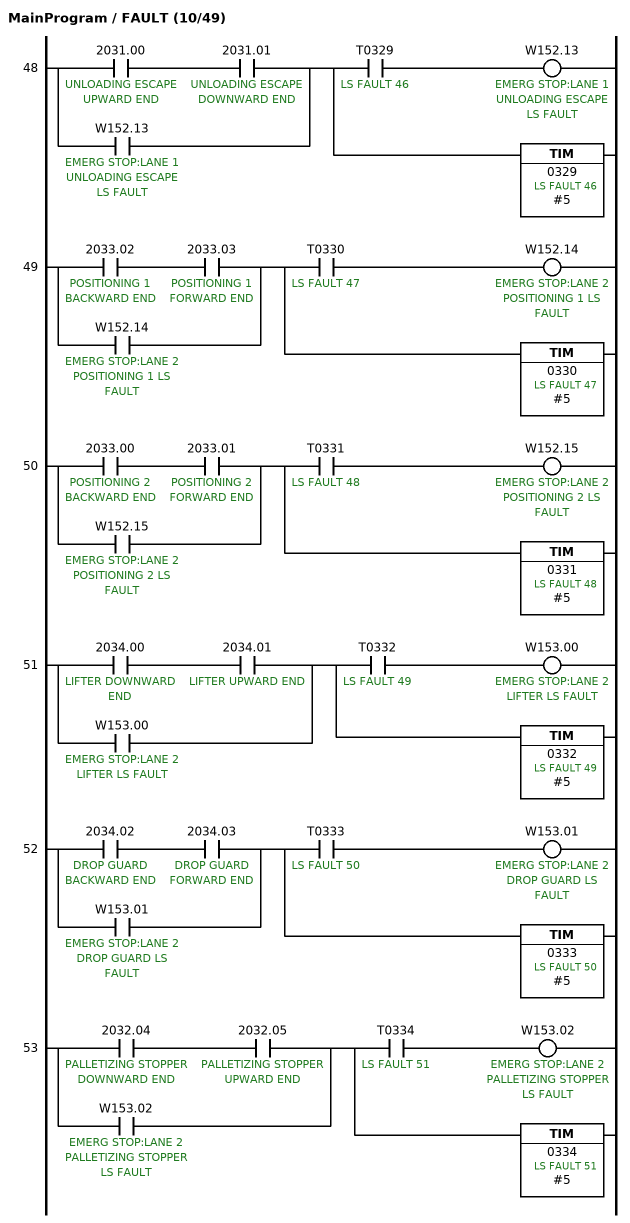
; [picture p72: MainProgram / FAULT, rungs 48-53]
; rung 48
LD 2031.00  ; UNLOADING ESCAPE UPWARD END
AND 2031.01  ; UNLOADING ESCAPE DOWNWARD END
OR W152.13  ; EMERG STOP:LANE 1 UNLOADING ESCAPE LS FAULT
OUT TR0
AND T0329  ; LS FAULT 46
OUT W152.13  ; EMERG STOP:LANE 1 UNLOADING ESCAPE LS FAULT
LD TR0
TIM 0329 #5  ; LS FAULT 46
; rung 49
LD 2033.02  ; POSITIONING 1 BACKWARD END
AND 2033.03  ; POSITIONING 1 FORWARD END
OR W152.14  ; EMERG STOP:LANE 2 POSITIONING 1 LS FAULT
OUT TR0
AND T0330  ; LS FAULT 47
OUT W152.14  ; EMERG STOP:LANE 2 POSITIONING 1 LS FAULT
LD TR0
TIM 0330 #5  ; LS FAULT 47
; rung 50
LD 2033.00  ; POSITIONING 2 BACKWARD END
AND 2033.01  ; POSITIONING 2 FORWARD END
OR W152.15  ; EMERG STOP:LANE 2 POSITIONING 2 LS FAULT
OUT TR0
AND T0331  ; LS FAULT 48
OUT W152.15  ; EMERG STOP:LANE 2 POSITIONING 2 LS FAULT
LD TR0
TIM 0331 #5  ; LS FAULT 48
; rung 51
LD 2034.00  ; LIFTER DOWNWARD END
AND 2034.01  ; LIFTER UPWARD END
OR W153.00  ; EMERG STOP:LANE 2 LIFTER LS FAULT
OUT TR0
AND T0332  ; LS FAULT 49
OUT W153.00  ; EMERG STOP:LANE 2 LIFTER LS FAULT
LD TR0
TIM 0332 #5  ; LS FAULT 49
; rung 52
LD 2034.02  ; DROP GUARD BACKWARD END
AND 2034.03  ; DROP GUARD FORWARD END
OR W153.01  ; EMERG STOP:LANE 2 DROP GUARD LS FAULT
OUT TR0
AND T0333  ; LS FAULT 50
OUT W153.01  ; EMERG STOP:LANE 2 DROP GUARD LS FAULT
LD TR0
TIM 0333 #5  ; LS FAULT 50
; rung 53
LD 2032.04  ; PALLETIZING STOPPER DOWNWARD END
AND 2032.05  ; PALLETIZING STOPPER UPWARD END
OR W153.02  ; EMERG STOP:LANE 2 PALLETIZING STOPPER LS FAULT
OUT TR0
AND T0334  ; LS FAULT 51
OUT W153.02  ; EMERG STOP:LANE 2 PALLETIZING STOPPER LS FAULT
LD TR0
TIM 0334 #5  ; LS FAULT 51

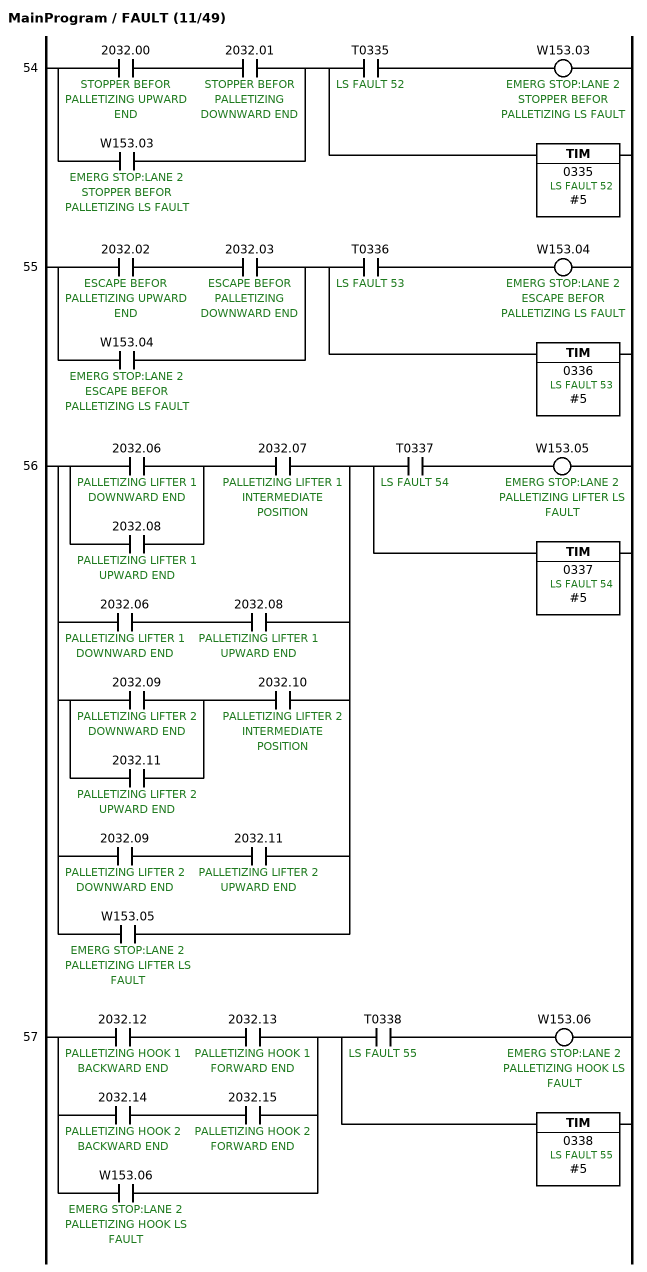
; rung 54
LD 2032.00  ; STOPPER BEFOR PALLETIZING UPWARD END
AND 2032.01  ; STOPPER BEFOR PALLETIZING DOWNWARD END
OR W153.03  ; EMERG STOP:LANE 2 STOPPER BEFOR PALLETIZING LS FAULT
OUT TR0
AND T0335  ; LS FAULT 52
OUT W153.03  ; EMERG STOP:LANE 2 STOPPER BEFOR PALLETIZING LS FAULT
LD TR0
TIM 0335 #5  ; LS FAULT 52
; rung 55
LD 2032.02  ; ESCAPE BEFOR PALLETIZING UPWARD END
AND 2032.03  ; ESCAPE BEFOR PALLETIZING DOWNWARD END
OR W153.04  ; EMERG STOP:LANE 2 ESCAPE BEFOR PALLETIZING LS FAULT
OUT TR0
AND T0336  ; LS FAULT 53
OUT W153.04  ; EMERG STOP:LANE 2 ESCAPE BEFOR PALLETIZING LS FAULT
LD TR0
TIM 0336 #5  ; LS FAULT 53
; rung 56
LD 2032.06  ; PALLETIZING LIFTER 1 DOWNWARD END
OR 2032.08  ; PALLETIZING LIFTER 1 UPWARD END
AND 2032.07  ; PALLETIZING LIFTER 1 INTERMEDIATE POSITION
LD 2032.06  ; PALLETIZING LIFTER 1 DOWNWARD END
AND 2032.08  ; PALLETIZING LIFTER 1 UPWARD END
ORLD
LD 2032.09  ; PALLETIZING LIFTER 2 DOWNWARD END
OR 2032.11  ; PALLETIZING LIFTER 2 UPWARD END
AND 2032.10  ; PALLETIZING LIFTER 2 INTERMEDIATE POSITION
ORLD
LD 2032.09  ; PALLETIZING LIFTER 2 DOWNWARD END
AND 2032.11  ; PALLETIZING LIFTER 2 UPWARD END
ORLD
OR W153.05  ; EMERG STOP:LANE 2 PALLETIZING LIFTER LS FAULT
OUT TR0
AND T0337  ; LS FAULT 54
OUT W153.05  ; EMERG STOP:LANE 2 PALLETIZING LIFTER LS FAULT
LD TR0
TIM 0337 #5  ; LS FAULT 54
; rung 57
LD 2032.12  ; PALLETIZING HOOK 1 BACKWARD END
AND 2032.13  ; PALLETIZING HOOK 1 FORWARD END
LD 2032.14  ; PALLETIZING HOOK 2 BACKWARD END
AND 2032.15  ; PALLETIZING HOOK 2 FORWARD END
ORLD
OR W153.06  ; EMERG STOP:LANE 2 PALLETIZING HOOK LS FAULT
OUT TR0
AND T0338  ; LS FAULT 55
OUT W153.06  ; EMERG STOP:LANE 2 PALLETIZING HOOK LS FAULT
LD TR0
TIM 0338 #5  ; LS FAULT 55

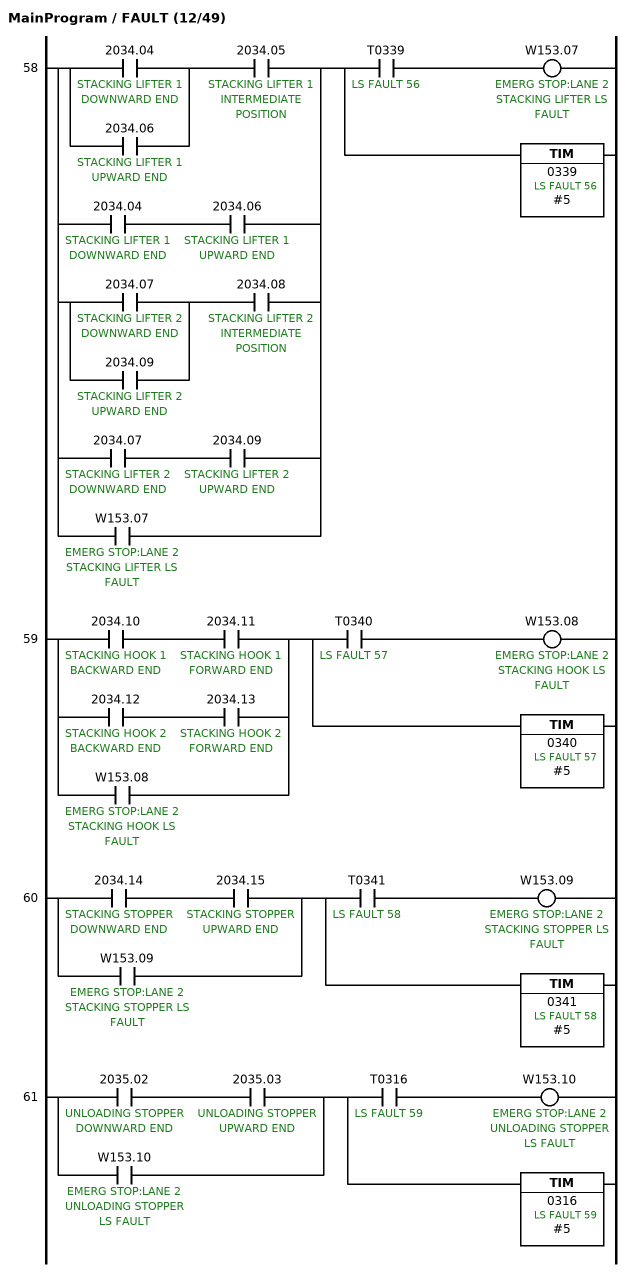
; rung 58
LD 2034.04  ; STACKING LIFTER 1 DOWNWARD END
OR 2034.06  ; STACKING LIFTER 1 UPWARD END
AND 2034.05  ; STACKING LIFTER 1 INTERMEDIATE POSITION
LD 2034.04  ; STACKING LIFTER 1 DOWNWARD END
AND 2034.06  ; STACKING LIFTER 1 UPWARD END
ORLD
LD 2034.07  ; STACKING LIFTER 2 DOWNWARD END
OR 2034.09  ; STACKING LIFTER 2 UPWARD END
AND 2034.08  ; STACKING LIFTER 2 INTERMEDIATE POSITION
ORLD
LD 2034.07  ; STACKING LIFTER 2 DOWNWARD END
AND 2034.09  ; STACKING LIFTER 2 UPWARD END
ORLD
OR W153.07  ; EMERG STOP:LANE 2 STACKING LIFTER LS FAULT
OUT TR0
AND T0339  ; LS FAULT 56
OUT W153.07  ; EMERG STOP:LANE 2 STACKING LIFTER LS FAULT
LD TR0
TIM 0339 #5  ; LS FAULT 56
; rung 59
LD 2034.10  ; STACKING HOOK 1 BACKWARD END
AND 2034.11  ; STACKING HOOK 1 FORWARD END
LD 2034.12  ; STACKING HOOK 2 BACKWARD END
AND 2034.13  ; STACKING HOOK 2 FORWARD END
ORLD
OR W153.08  ; EMERG STOP:LANE 2 STACKING HOOK LS FAULT
OUT TR0
AND T0340  ; LS FAULT 57
OUT W153.08  ; EMERG STOP:LANE 2 STACKING HOOK LS FAULT
LD TR0
TIM 0340 #5  ; LS FAULT 57
; rung 60
LD 2034.14  ; STACKING STOPPER DOWNWARD END
AND 2034.15  ; STACKING STOPPER UPWARD END
OR W153.09  ; EMERG STOP:LANE 2 STACKING STOPPER LS FAULT
OUT TR0
AND T0341  ; LS FAULT 58
OUT W153.09  ; EMERG STOP:LANE 2 STACKING STOPPER LS FAULT
LD TR0
TIM 0341 #5  ; LS FAULT 58
; rung 61
LD 2035.02  ; UNLOADING STOPPER DOWNWARD END
AND 2035.03  ; UNLOADING STOPPER UPWARD END
OR W153.10  ; EMERG STOP:LANE 2 UNLOADING STOPPER LS FAULT
OUT TR0
AND T0316  ; LS FAULT 59
OUT W153.10  ; EMERG STOP:LANE 2 UNLOADING STOPPER LS FAULT
LD TR0
TIM 0316 #5  ; LS FAULT 59

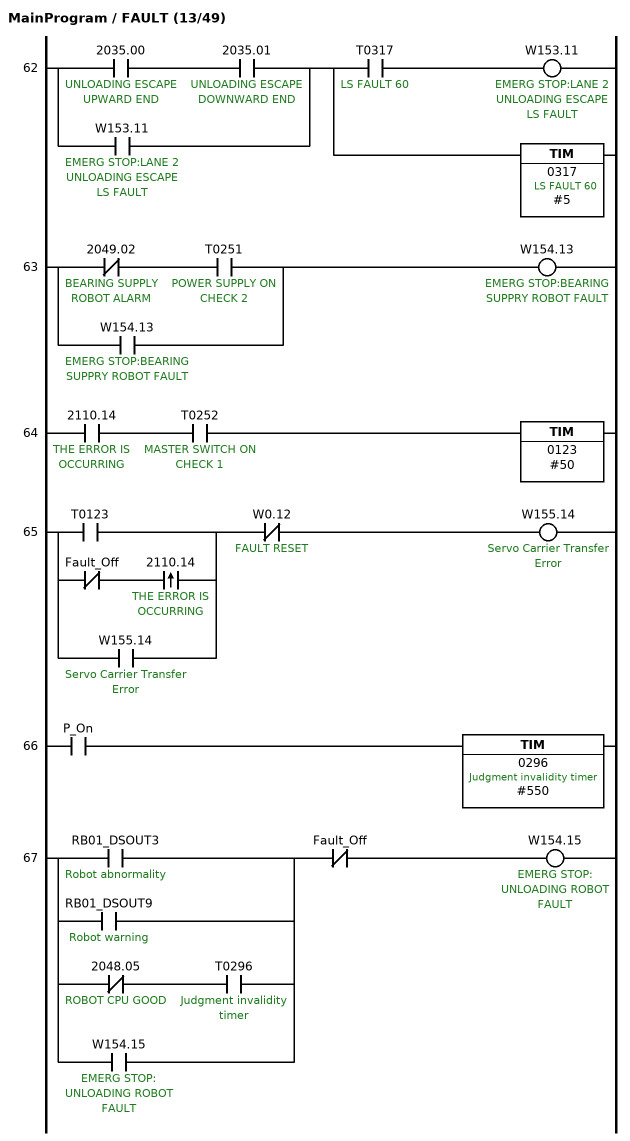
; rung 62
LD 2035.00  ; UNLOADING ESCAPE UPWARD END
AND 2035.01  ; UNLOADING ESCAPE DOWNWARD END
OR W153.11  ; EMERG STOP:LANE 2 UNLOADING ESCAPE LS FAULT
OUT TR0
AND T0317  ; LS FAULT 60
OUT W153.11  ; EMERG STOP:LANE 2 UNLOADING ESCAPE LS FAULT
LD TR0
TIM 0317 #5  ; LS FAULT 60
; rung 63
LDNOT 2049.02  ; BEARING SUPPLY ROBOT ALARM
AND T0251  ; POWER SUPPLY ON CHECK 2
OR W154.13  ; EMERG STOP:BEARING SUPPRY ROBOT FAULT
OUT W154.13  ; EMERG STOP:BEARING SUPPRY ROBOT FAULT
; rung 64
LD 2110.14  ; THE ERROR IS OCCURRING
AND T0252  ; MASTER SWITCH ON CHECK 1
TIM 0123 #50
; rung 65
LD T0123
LDNOT Fault_Off
@AND 2110.14  ; THE ERROR IS OCCURRING
ORLD
OR W155.14  ; Servo Carrier Transfer Error
ANDNOT W0.12  ; FAULT RESET
OUT W155.14  ; Servo Carrier Transfer Error
; rung 66
LD P_On
TIM 0296 #550  ; Judgment invalidity timer
; rung 67
LD RB01_DSOUT3  ; Robot abnormality
OR RB01_DSOUT9  ; Robot warning
LDNOT 2048.05  ; ROBOT CPU GOOD
AND T0296  ; Judgment invalidity timer
ORLD
OR W154.15  ; EMERG STOP:UNLOADING ROBOT FAULT
ANDNOT Fault_Off
OUT W154.15  ; EMERG STOP:UNLOADING ROBOT FAULT

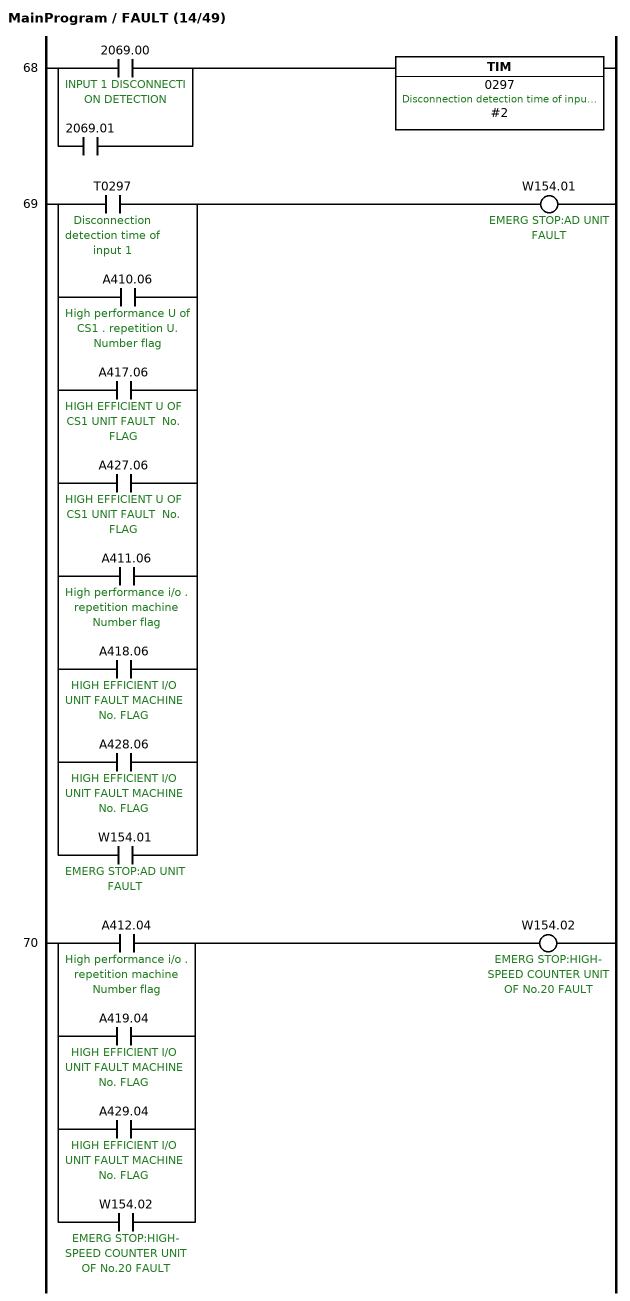
; rung 68
LD 2069.00  ; INPUT 1 DISCONNECTION DETECTION
OR 2069.01
TIM 0297 #2  ; Disconnection detection time of input 1
; rung 69
LD T0297  ; Disconnection detection time of input 1
OR A410.06  ; High performance U of CS1 . repetition U. Number flag
OR A417.06  ; HIGH EFFICIENT U OF CS1 UNIT FAULT  No. FLAG
OR A427.06  ; HIGH EFFICIENT U OF CS1 UNIT FAULT  No. FLAG
OR A411.06  ; High performance i/o . repetition machine Number flag
OR A418.06  ; HIGH EFFICIENT I/O UNIT FAULT MACHINE No. FLAG
OR A428.06  ; HIGH EFFICIENT I/O UNIT FAULT MACHINE No. FLAG
OR W154.01  ; EMERG STOP:AD UNIT FAULT
OUT W154.01  ; EMERG STOP:AD UNIT FAULT
; rung 70
LD A412.04  ; High performance i/o . repetition machine Number flag
OR A419.04  ; HIGH EFFICIENT I/O UNIT FAULT MACHINE No. FLAG
OR A429.04  ; HIGH EFFICIENT I/O UNIT FAULT MACHINE No. FLAG
OR W154.02  ; EMERG STOP:HIGH-SPEED COUNTER UNIT OF No.20 FAULT
OUT W154.02  ; EMERG STOP:HIGH-SPEED COUNTER UNIT OF No.20 FAULT

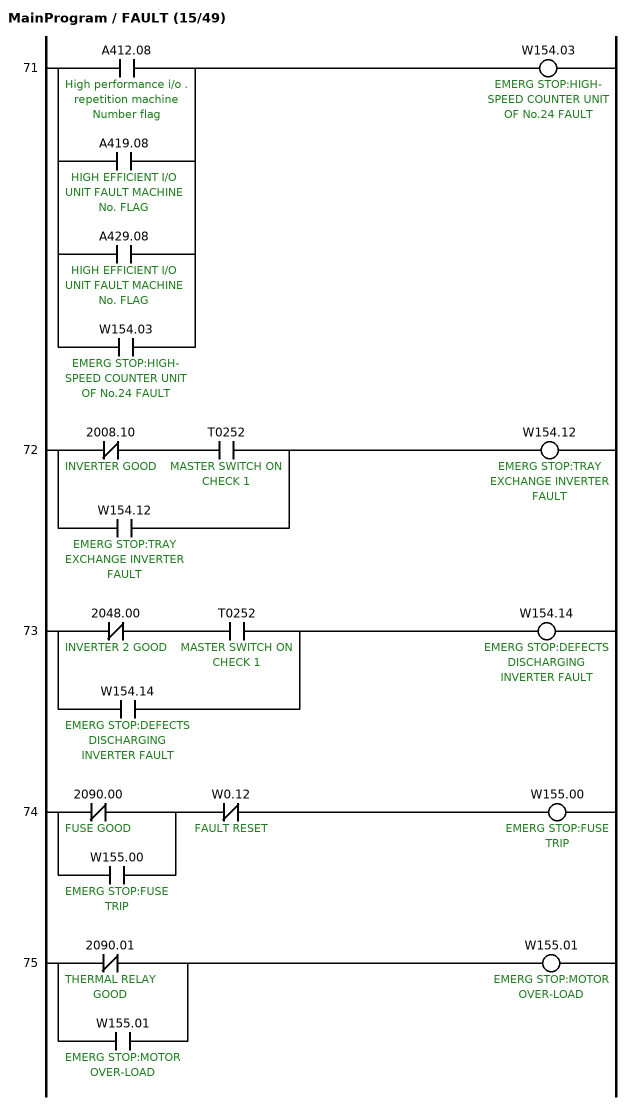
; rung 71
LD A412.08  ; High performance i/o . repetition machine Number flag
OR A419.08  ; HIGH EFFICIENT I/O UNIT FAULT MACHINE No. FLAG
OR A429.08  ; HIGH EFFICIENT I/O UNIT FAULT MACHINE No. FLAG
OR W154.03  ; EMERG STOP:HIGH-SPEED COUNTER UNIT OF No.24 FAULT
OUT W154.03  ; EMERG STOP:HIGH-SPEED COUNTER UNIT OF No.24 FAULT
; rung 72
LDNOT 2008.10  ; INVERTER GOOD
AND T0252  ; MASTER SWITCH ON CHECK 1
OR W154.12  ; EMERG STOP:TRAY EXCHANGE INVERTER FAULT
OUT W154.12  ; EMERG STOP:TRAY EXCHANGE INVERTER FAULT
; rung 73
LDNOT 2048.00  ; INVERTER 2 GOOD
AND T0252  ; MASTER SWITCH ON CHECK 1
OR W154.14  ; EMERG STOP:DEFECTS DISCHARGING INVERTER FAULT
OUT W154.14  ; EMERG STOP:DEFECTS DISCHARGING INVERTER FAULT
; rung 74
LDNOT 2090.00  ; FUSE GOOD
OR W155.00  ; EMERG STOP:FUSE TRIP
ANDNOT W0.12  ; FAULT RESET
OUT W155.00  ; EMERG STOP:FUSE TRIP
; rung 75
LDNOT 2090.01  ; THERMAL RELAY GOOD
OR W155.01  ; EMERG STOP:MOTOR OVER-LOAD
OUT W155.01  ; EMERG STOP:MOTOR OVER-LOAD

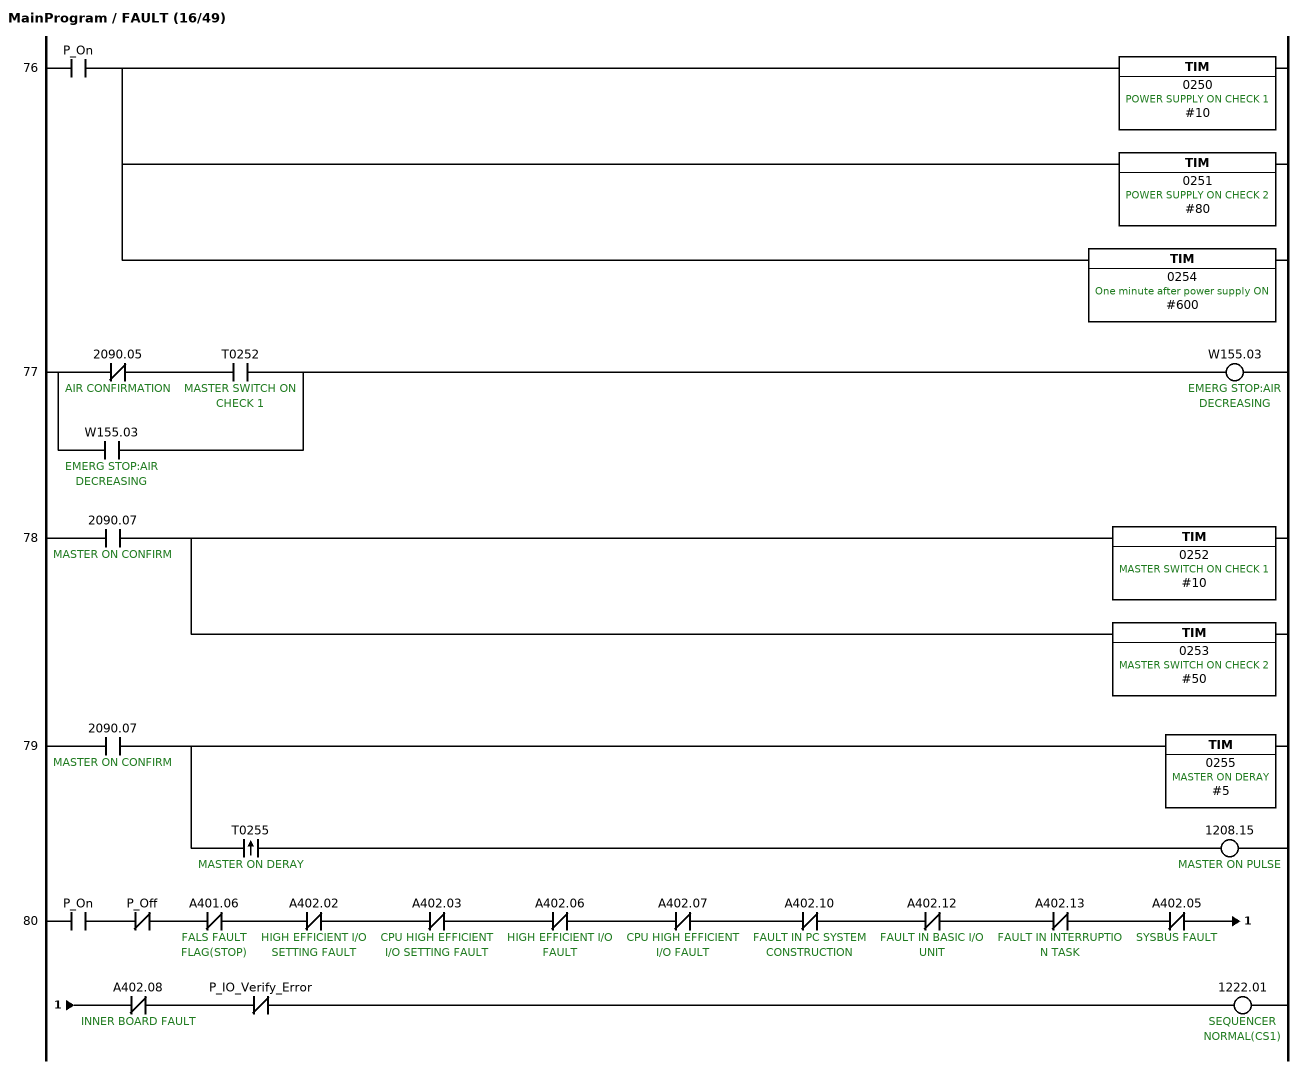
; rung 76
LD P_On
TIM 0250 #10  ; POWER SUPPLY ON CHECK 1
TIM 0251 #80  ; POWER SUPPLY ON CHECK 2
TIM 0254 #600  ; One minute after power supply ON
; rung 77
LDNOT 2090.05  ; AIR CONFIRMATION
AND T0252  ; MASTER SWITCH ON CHECK 1
OR W155.03  ; EMERG STOP:AIR DECREASING
OUT W155.03  ; EMERG STOP:AIR DECREASING
; rung 78
LD 2090.07  ; MASTER ON CONFIRM
TIM 0252 #10  ; MASTER SWITCH ON CHECK 1
TIM 0253 #50  ; MASTER SWITCH ON CHECK 2
; rung 79
LD 2090.07  ; MASTER ON CONFIRM
TIM 0255 #5  ; MASTER ON DERAY
@AND T0255  ; MASTER ON DERAY
OUT 1208.15  ; MASTER ON PULSE
; rung 80
LD P_On
ANDNOT P_Off
ANDNOT A401.06  ; FALS FAULT FLAG(STOP)
ANDNOT A402.02  ; HIGH EFFICIENT I/O SETTING FAULT
ANDNOT A402.03  ; CPU HIGH EFFICIENT I/O SETTING FAULT
ANDNOT A402.06  ; HIGH EFFICIENT I/O FAULT
ANDNOT A402.07  ; CPU HIGH EFFICIENT I/O FAULT
ANDNOT A402.10  ; FAULT IN PC SYSTEM CONSTRUCTION
ANDNOT A402.12  ; FAULT IN BASIC I/O UNIT
ANDNOT A402.13  ; FAULT IN INTERRUPTION TASK
ANDNOT A402.05  ; SYSBUS FAULT
ANDNOT A402.08  ; INNER BOARD FAULT
ANDNOT P_IO_Verify_Error
OUT 1222.01  ; SEQUENCER NORMAL(CS1)

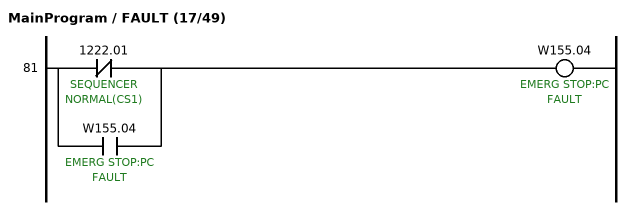
; rung 81
LDNOT 1222.01  ; SEQUENCER NORMAL(CS1)
OR W155.04  ; EMERG STOP:PC FAULT
OUT W155.04  ; EMERG STOP:PC FAULT

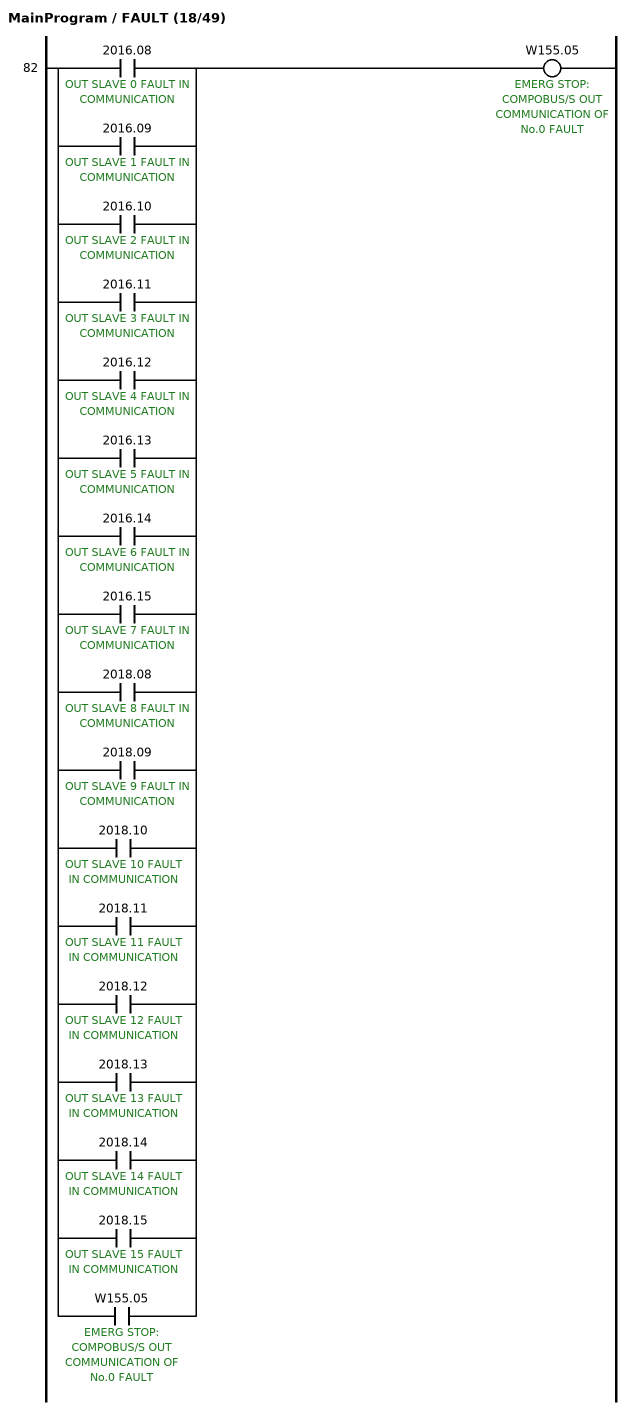
; rung 82
LD 2016.08  ; OUT SLAVE 0 FAULT IN COMMUNICATION
OR 2016.09  ; OUT SLAVE 1 FAULT IN COMMUNICATION
OR 2016.10  ; OUT SLAVE 2 FAULT IN COMMUNICATION
OR 2016.11  ; OUT SLAVE 3 FAULT IN COMMUNICATION
OR 2016.12  ; OUT SLAVE 4 FAULT IN COMMUNICATION
OR 2016.13  ; OUT SLAVE 5 FAULT IN COMMUNICATION
OR 2016.14  ; OUT SLAVE 6 FAULT IN COMMUNICATION
OR 2016.15  ; OUT SLAVE 7 FAULT IN COMMUNICATION
OR 2018.08  ; OUT SLAVE 8 FAULT IN COMMUNICATION
OR 2018.09  ; OUT SLAVE 9 FAULT IN COMMUNICATION
OR 2018.10  ; OUT SLAVE 10 FAULT IN COMMUNICATION
OR 2018.11  ; OUT SLAVE 11 FAULT IN COMMUNICATION
OR 2018.12  ; OUT SLAVE 12 FAULT IN COMMUNICATION
OR 2018.13  ; OUT SLAVE 13 FAULT IN COMMUNICATION
OR 2018.14  ; OUT SLAVE 14 FAULT IN COMMUNICATION
OR 2018.15  ; OUT SLAVE 15 FAULT IN COMMUNICATION
OR W155.05  ; EMERG STOP:COMPOBUS/S OUT COMMUNICATION OF No.0 FAULT
OUT W155.05  ; EMERG STOP:COMPOBUS/S OUT COMMUNICATION OF No.0 FAULT

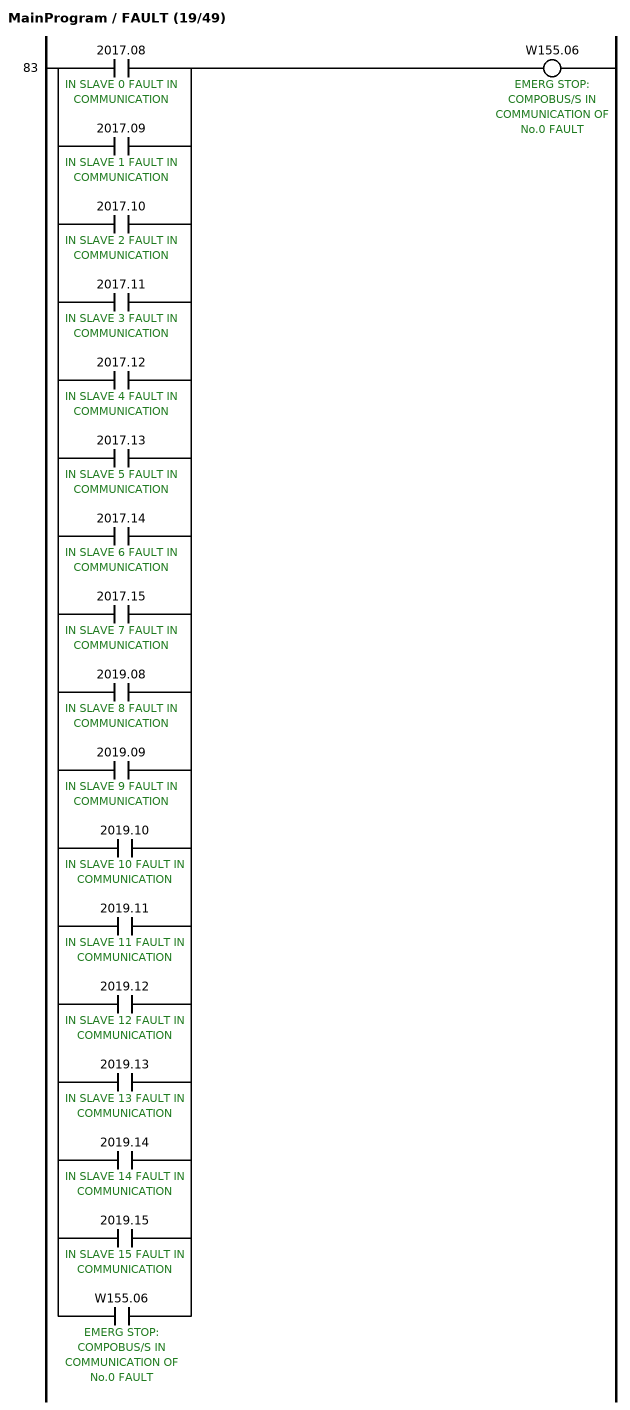
; rung 83
LD 2017.08  ; IN SLAVE 0 FAULT IN COMMUNICATION
OR 2017.09  ; IN SLAVE 1 FAULT IN COMMUNICATION
OR 2017.10  ; IN SLAVE 2 FAULT IN COMMUNICATION
OR 2017.11  ; IN SLAVE 3 FAULT IN COMMUNICATION
OR 2017.12  ; IN SLAVE 4 FAULT IN COMMUNICATION
OR 2017.13  ; IN SLAVE 5 FAULT IN COMMUNICATION
OR 2017.14  ; IN SLAVE 6 FAULT IN COMMUNICATION
OR 2017.15  ; IN SLAVE 7 FAULT IN COMMUNICATION
OR 2019.08  ; IN SLAVE 8 FAULT IN COMMUNICATION
OR 2019.09  ; IN SLAVE 9 FAULT IN COMMUNICATION
OR 2019.10  ; IN SLAVE 10 FAULT IN COMMUNICATION
OR 2019.11  ; IN SLAVE 11 FAULT IN COMMUNICATION
OR 2019.12  ; IN SLAVE 12 FAULT IN COMMUNICATION
OR 2019.13  ; IN SLAVE 13 FAULT IN COMMUNICATION
OR 2019.14  ; IN SLAVE 14 FAULT IN COMMUNICATION
OR 2019.15  ; IN SLAVE 15 FAULT IN COMMUNICATION
OR W155.06  ; EMERG STOP:COMPOBUS/S IN COMMUNICATION OF No.0 FAULT
OUT W155.06  ; EMERG STOP:COMPOBUS/S IN COMMUNICATION OF No.0 FAULT

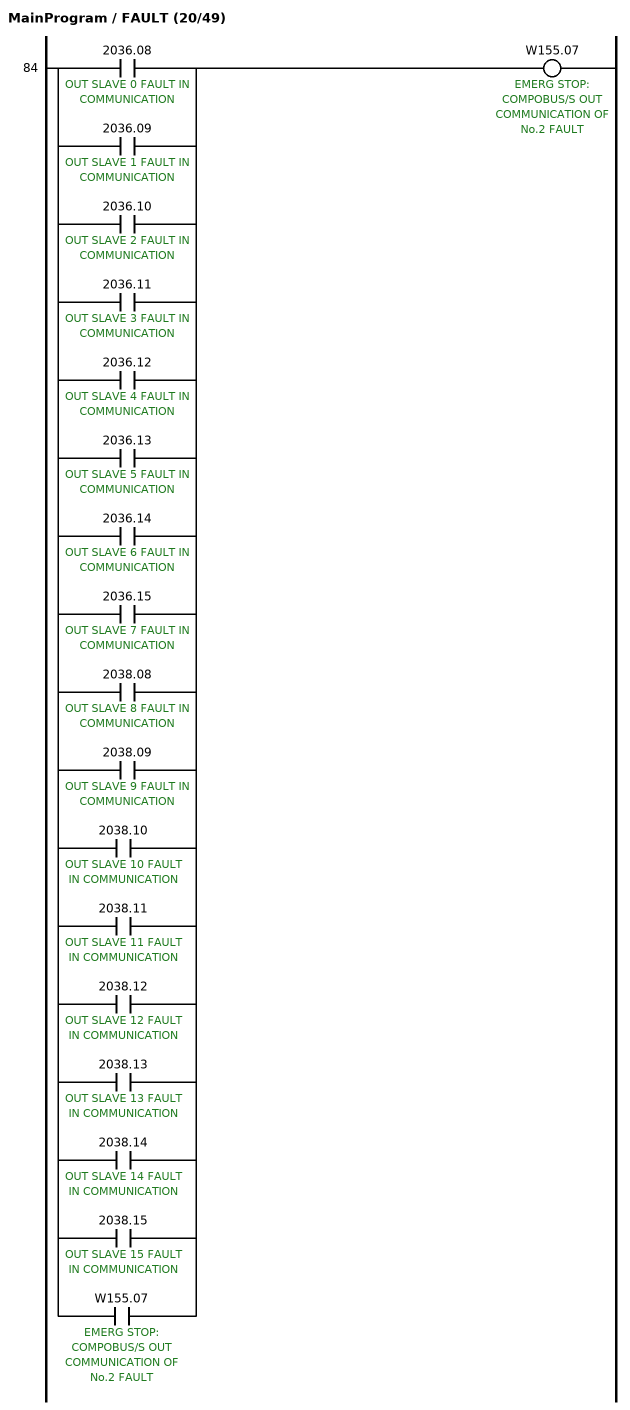
; rung 84
LD 2036.08  ; OUT SLAVE 0 FAULT IN COMMUNICATION
OR 2036.09  ; OUT SLAVE 1 FAULT IN COMMUNICATION
OR 2036.10  ; OUT SLAVE 2 FAULT IN COMMUNICATION
OR 2036.11  ; OUT SLAVE 3 FAULT IN COMMUNICATION
OR 2036.12  ; OUT SLAVE 4 FAULT IN COMMUNICATION
OR 2036.13  ; OUT SLAVE 5 FAULT IN COMMUNICATION
OR 2036.14  ; OUT SLAVE 6 FAULT IN COMMUNICATION
OR 2036.15  ; OUT SLAVE 7 FAULT IN COMMUNICATION
OR 2038.08  ; OUT SLAVE 8 FAULT IN COMMUNICATION
OR 2038.09  ; OUT SLAVE 9 FAULT IN COMMUNICATION
OR 2038.10  ; OUT SLAVE 10 FAULT IN COMMUNICATION
OR 2038.11  ; OUT SLAVE 11 FAULT IN COMMUNICATION
OR 2038.12  ; OUT SLAVE 12 FAULT IN COMMUNICATION
OR 2038.13  ; OUT SLAVE 13 FAULT IN COMMUNICATION
OR 2038.14  ; OUT SLAVE 14 FAULT IN COMMUNICATION
OR 2038.15  ; OUT SLAVE 15 FAULT IN COMMUNICATION
OR W155.07  ; EMERG STOP:COMPOBUS/S OUT COMMUNICATION OF No.2 FAULT
OUT W155.07  ; EMERG STOP:COMPOBUS/S OUT COMMUNICATION OF No.2 FAULT

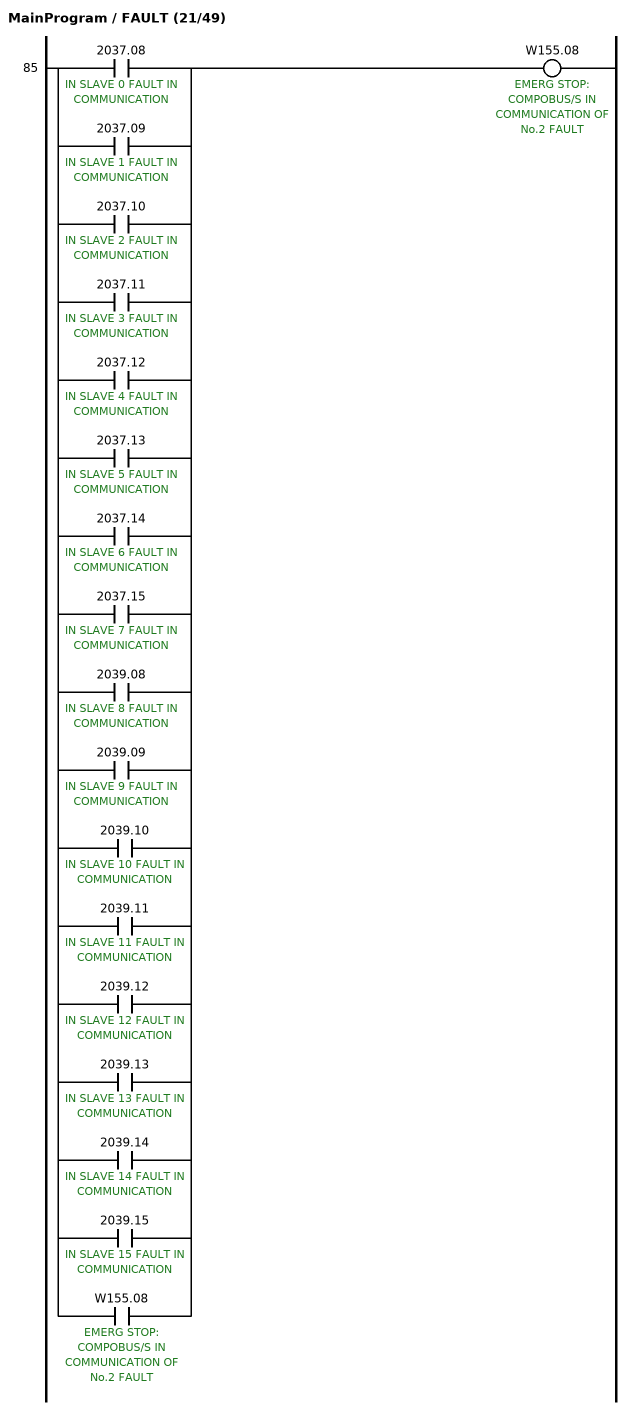
; rung 85
LD 2037.08  ; IN SLAVE 0 FAULT IN COMMUNICATION
OR 2037.09  ; IN SLAVE 1 FAULT IN COMMUNICATION
OR 2037.10  ; IN SLAVE 2 FAULT IN COMMUNICATION
OR 2037.11  ; IN SLAVE 3 FAULT IN COMMUNICATION
OR 2037.12  ; IN SLAVE 4 FAULT IN COMMUNICATION
OR 2037.13  ; IN SLAVE 5 FAULT IN COMMUNICATION
OR 2037.14  ; IN SLAVE 6 FAULT IN COMMUNICATION
OR 2037.15  ; IN SLAVE 7 FAULT IN COMMUNICATION
OR 2039.08  ; IN SLAVE 8 FAULT IN COMMUNICATION
OR 2039.09  ; IN SLAVE 9 FAULT IN COMMUNICATION
OR 2039.10  ; IN SLAVE 10 FAULT IN COMMUNICATION
OR 2039.11  ; IN SLAVE 11 FAULT IN COMMUNICATION
OR 2039.12  ; IN SLAVE 12 FAULT IN COMMUNICATION
OR 2039.13  ; IN SLAVE 13 FAULT IN COMMUNICATION
OR 2039.14  ; IN SLAVE 14 FAULT IN COMMUNICATION
OR 2039.15  ; IN SLAVE 15 FAULT IN COMMUNICATION
OR W155.08  ; EMERG STOP:COMPOBUS/S IN COMMUNICATION OF No.2 FAULT
OUT W155.08  ; EMERG STOP:COMPOBUS/S IN COMMUNICATION OF No.2 FAULT

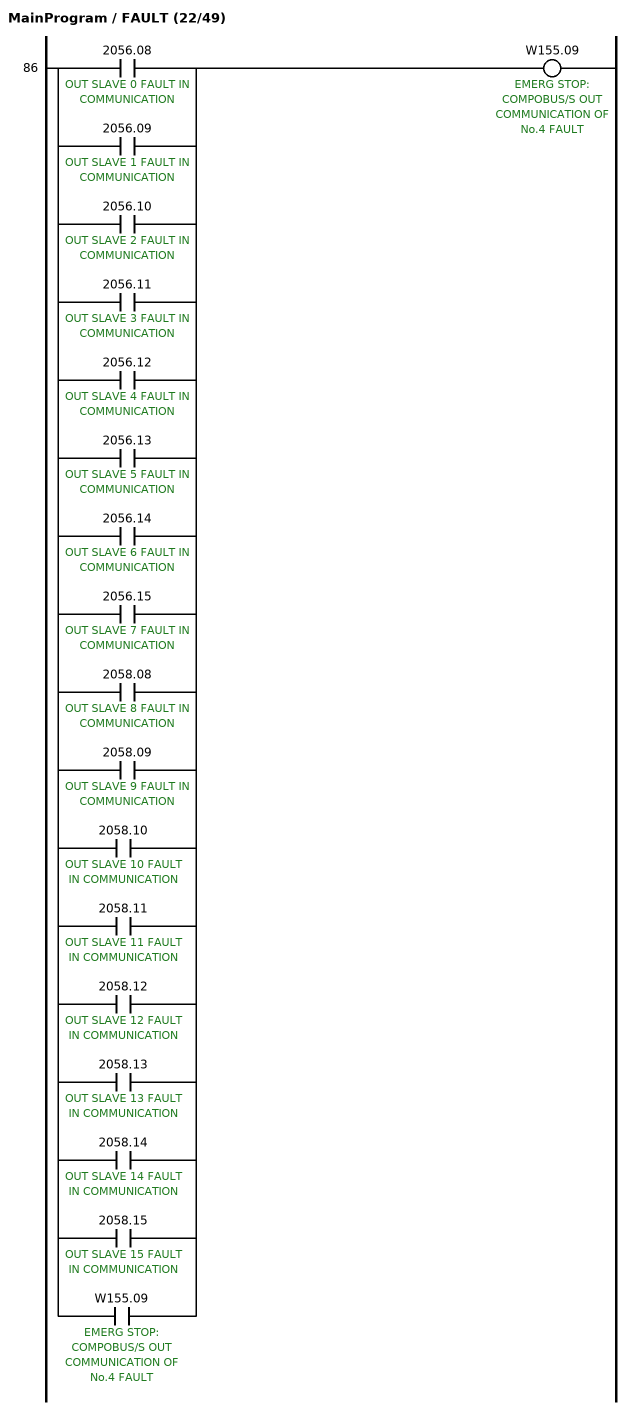
; rung 86
LD 2056.08  ; OUT SLAVE 0 FAULT IN COMMUNICATION
OR 2056.09  ; OUT SLAVE 1 FAULT IN COMMUNICATION
OR 2056.10  ; OUT SLAVE 2 FAULT IN COMMUNICATION
OR 2056.11  ; OUT SLAVE 3 FAULT IN COMMUNICATION
OR 2056.12  ; OUT SLAVE 4 FAULT IN COMMUNICATION
OR 2056.13  ; OUT SLAVE 5 FAULT IN COMMUNICATION
OR 2056.14  ; OUT SLAVE 6 FAULT IN COMMUNICATION
OR 2056.15  ; OUT SLAVE 7 FAULT IN COMMUNICATION
OR 2058.08  ; OUT SLAVE 8 FAULT IN COMMUNICATION
OR 2058.09  ; OUT SLAVE 9 FAULT IN COMMUNICATION
OR 2058.10  ; OUT SLAVE 10 FAULT IN COMMUNICATION
OR 2058.11  ; OUT SLAVE 11 FAULT IN COMMUNICATION
OR 2058.12  ; OUT SLAVE 12 FAULT IN COMMUNICATION
OR 2058.13  ; OUT SLAVE 13 FAULT IN COMMUNICATION
OR 2058.14  ; OUT SLAVE 14 FAULT IN COMMUNICATION
OR 2058.15  ; OUT SLAVE 15 FAULT IN COMMUNICATION
OR W155.09  ; EMERG STOP:COMPOBUS/S OUT COMMUNICATION OF No.4 FAULT
OUT W155.09  ; EMERG STOP:COMPOBUS/S OUT COMMUNICATION OF No.4 FAULT

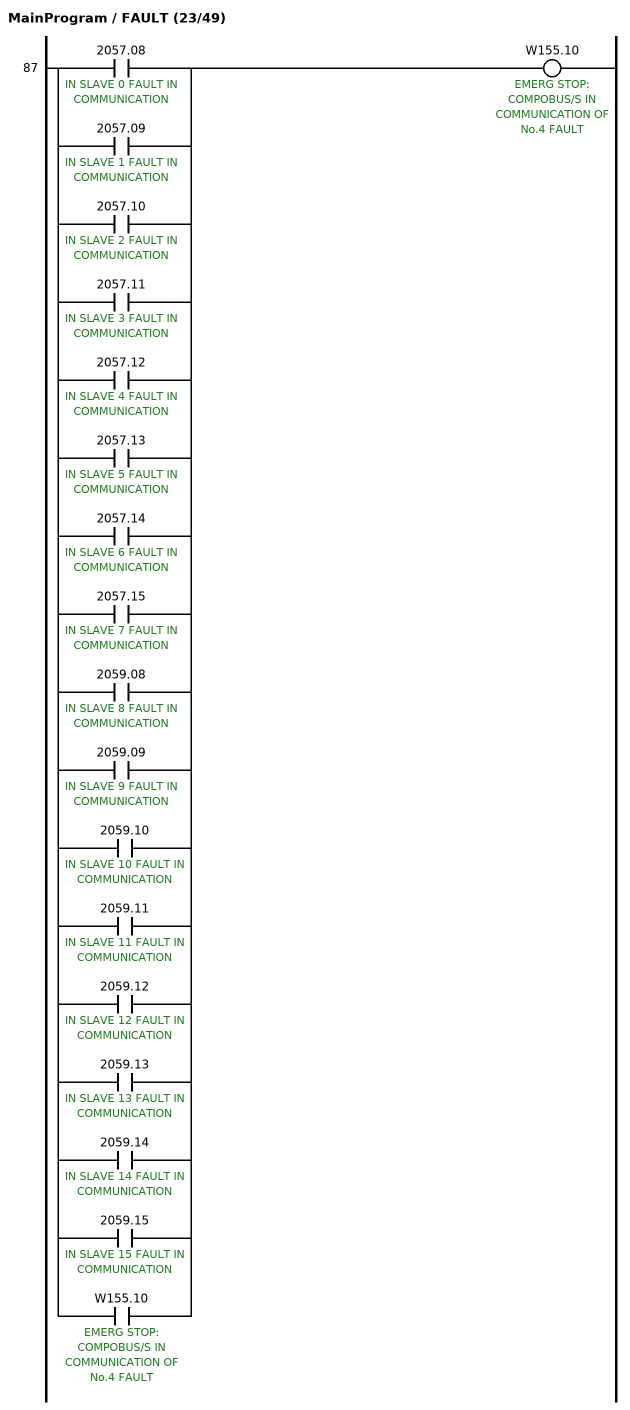
; rung 87
LD 2057.08  ; IN SLAVE 0 FAULT IN COMMUNICATION
OR 2057.09  ; IN SLAVE 1 FAULT IN COMMUNICATION
OR 2057.10  ; IN SLAVE 2 FAULT IN COMMUNICATION
OR 2057.11  ; IN SLAVE 3 FAULT IN COMMUNICATION
OR 2057.12  ; IN SLAVE 4 FAULT IN COMMUNICATION
OR 2057.13  ; IN SLAVE 5 FAULT IN COMMUNICATION
OR 2057.14  ; IN SLAVE 6 FAULT IN COMMUNICATION
OR 2057.15  ; IN SLAVE 7 FAULT IN COMMUNICATION
OR 2059.08  ; IN SLAVE 8 FAULT IN COMMUNICATION
OR 2059.09  ; IN SLAVE 9 FAULT IN COMMUNICATION
OR 2059.10  ; IN SLAVE 10 FAULT IN COMMUNICATION
OR 2059.11  ; IN SLAVE 11 FAULT IN COMMUNICATION
OR 2059.12  ; IN SLAVE 12 FAULT IN COMMUNICATION
OR 2059.13  ; IN SLAVE 13 FAULT IN COMMUNICATION
OR 2059.14  ; IN SLAVE 14 FAULT IN COMMUNICATION
OR 2059.15  ; IN SLAVE 15 FAULT IN COMMUNICATION
OR W155.10  ; EMERG STOP:COMPOBUS/S IN COMMUNICATION OF No.4 FAULT
OUT W155.10  ; EMERG STOP:COMPOBUS/S IN COMMUNICATION OF No.4 FAULT

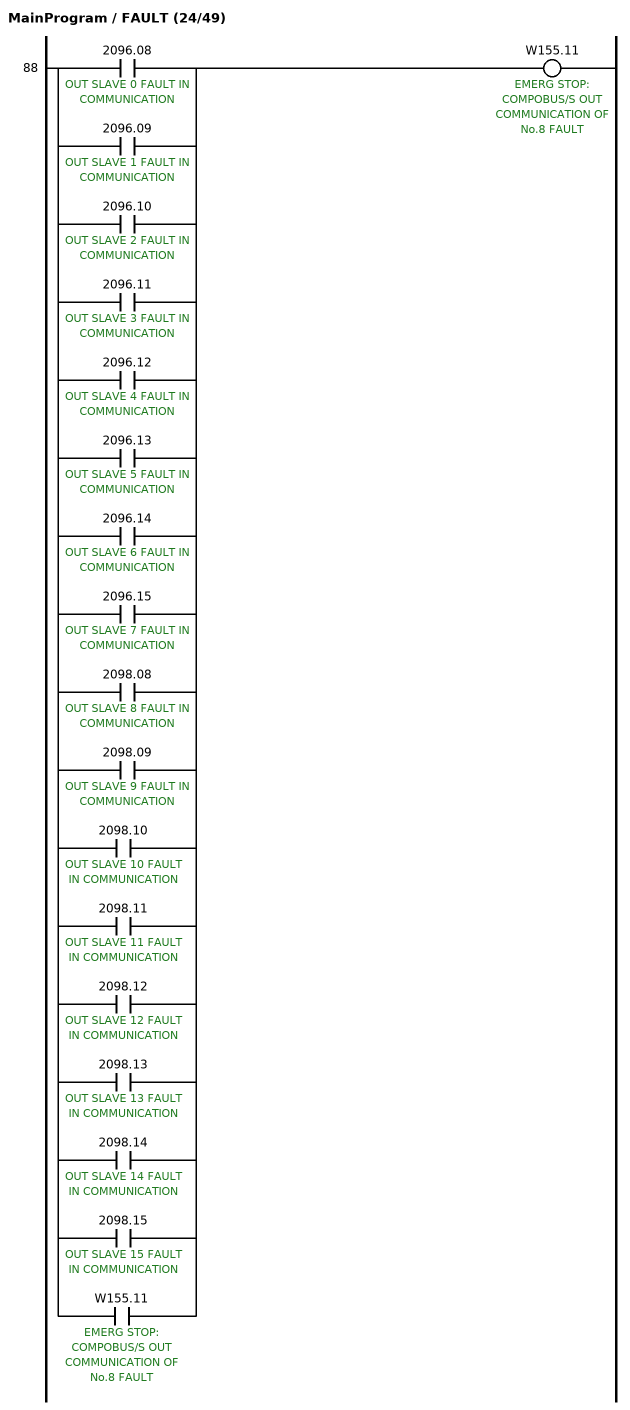
; rung 88
LD 2096.08  ; OUT SLAVE 0 FAULT IN COMMUNICATION
OR 2096.09  ; OUT SLAVE 1 FAULT IN COMMUNICATION
OR 2096.10  ; OUT SLAVE 2 FAULT IN COMMUNICATION
OR 2096.11  ; OUT SLAVE 3 FAULT IN COMMUNICATION
OR 2096.12  ; OUT SLAVE 4 FAULT IN COMMUNICATION
OR 2096.13  ; OUT SLAVE 5 FAULT IN COMMUNICATION
OR 2096.14  ; OUT SLAVE 6 FAULT IN COMMUNICATION
OR 2096.15  ; OUT SLAVE 7 FAULT IN COMMUNICATION
OR 2098.08  ; OUT SLAVE 8 FAULT IN COMMUNICATION
OR 2098.09  ; OUT SLAVE 9 FAULT IN COMMUNICATION
OR 2098.10  ; OUT SLAVE 10 FAULT IN COMMUNICATION
OR 2098.11  ; OUT SLAVE 11 FAULT IN COMMUNICATION
OR 2098.12  ; OUT SLAVE 12 FAULT IN COMMUNICATION
OR 2098.13  ; OUT SLAVE 13 FAULT IN COMMUNICATION
OR 2098.14  ; OUT SLAVE 14 FAULT IN COMMUNICATION
OR 2098.15  ; OUT SLAVE 15 FAULT IN COMMUNICATION
OR W155.11  ; EMERG STOP:COMPOBUS/S OUT COMMUNICATION OF No.8 FAULT
OUT W155.11  ; EMERG STOP:COMPOBUS/S OUT COMMUNICATION OF No.8 FAULT

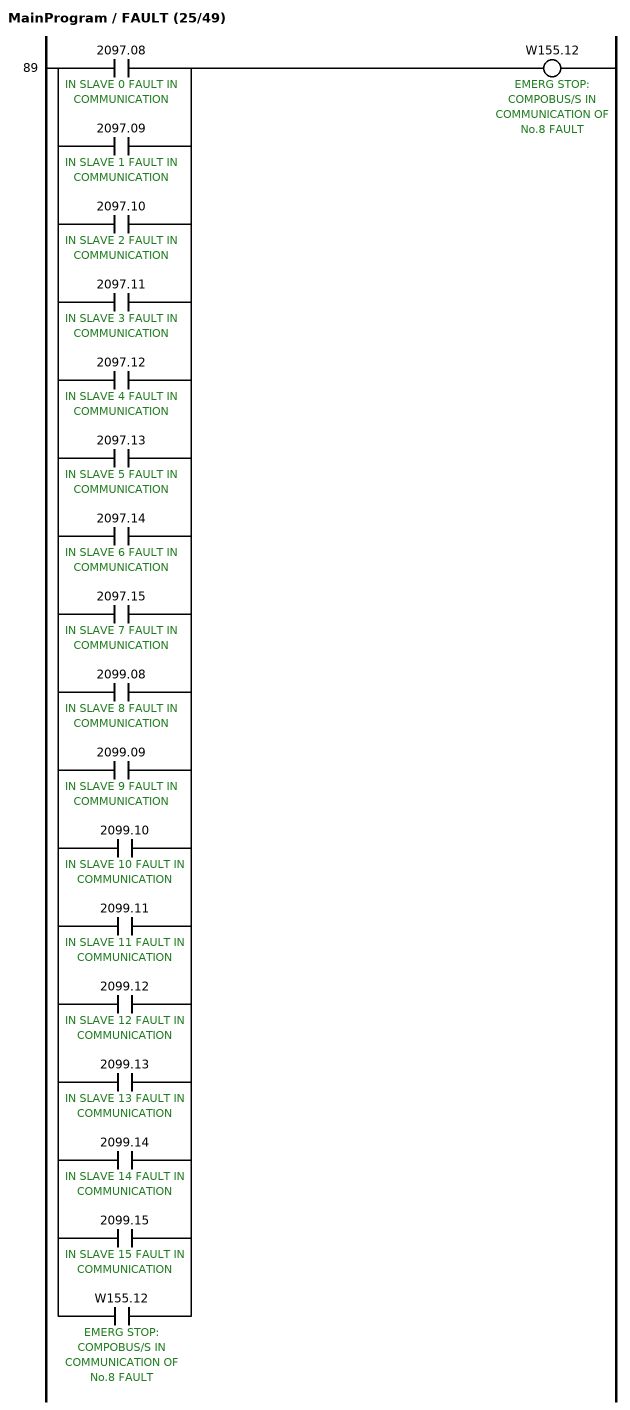
; rung 89
LD 2097.08  ; IN SLAVE 0 FAULT IN COMMUNICATION
OR 2097.09  ; IN SLAVE 1 FAULT IN COMMUNICATION
OR 2097.10  ; IN SLAVE 2 FAULT IN COMMUNICATION
OR 2097.11  ; IN SLAVE 3 FAULT IN COMMUNICATION
OR 2097.12  ; IN SLAVE 4 FAULT IN COMMUNICATION
OR 2097.13  ; IN SLAVE 5 FAULT IN COMMUNICATION
OR 2097.14  ; IN SLAVE 6 FAULT IN COMMUNICATION
OR 2097.15  ; IN SLAVE 7 FAULT IN COMMUNICATION
OR 2099.08  ; IN SLAVE 8 FAULT IN COMMUNICATION
OR 2099.09  ; IN SLAVE 9 FAULT IN COMMUNICATION
OR 2099.10  ; IN SLAVE 10 FAULT IN COMMUNICATION
OR 2099.11  ; IN SLAVE 11 FAULT IN COMMUNICATION
OR 2099.12  ; IN SLAVE 12 FAULT IN COMMUNICATION
OR 2099.13  ; IN SLAVE 13 FAULT IN COMMUNICATION
OR 2099.14  ; IN SLAVE 14 FAULT IN COMMUNICATION
OR 2099.15  ; IN SLAVE 15 FAULT IN COMMUNICATION
OR W155.12  ; EMERG STOP:COMPOBUS/S IN COMMUNICATION OF No.8 FAULT
OUT W155.12  ; EMERG STOP:COMPOBUS/S IN COMMUNICATION OF No.8 FAULT

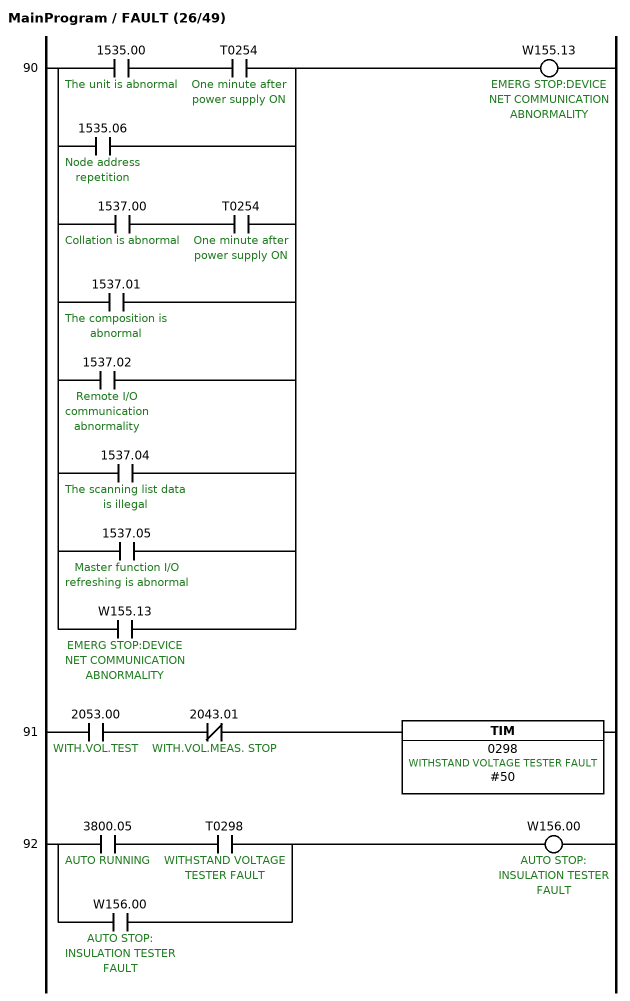
; rung 90
LD 1535.00  ; The unit is abnormal
AND T0254  ; One minute after power supply ON
OR 1535.06  ; Node address repetition
LD 1537.00  ; Collation is abnormal
AND T0254  ; One minute after power supply ON
ORLD
OR 1537.01  ; The composition is abnormal
OR 1537.02  ; Remote I/O communication abnormality
OR 1537.04  ; The scanning list data is illegal
OR 1537.05  ; Master function I/O refreshing is abnormal
OR W155.13  ; EMERG STOP:DEVICE NET COMMUNICATION ABNORMALITY
OUT W155.13  ; EMERG STOP:DEVICE NET COMMUNICATION ABNORMALITY
; rung 91
LD 2053.00  ; WITH.VOL.TEST
ANDNOT 2043.01  ; WITH.VOL.MEAS. STOP
TIM 0298 #50  ; WITHSTAND VOLTAGE TESTER FAULT
; rung 92
LD 3800.05  ; AUTO RUNNING
AND T0298  ; WITHSTAND VOLTAGE TESTER FAULT
OR W156.00  ; AUTO STOP:INSULATION TESTER FAULT
OUT W156.00  ; AUTO STOP:INSULATION TESTER FAULT

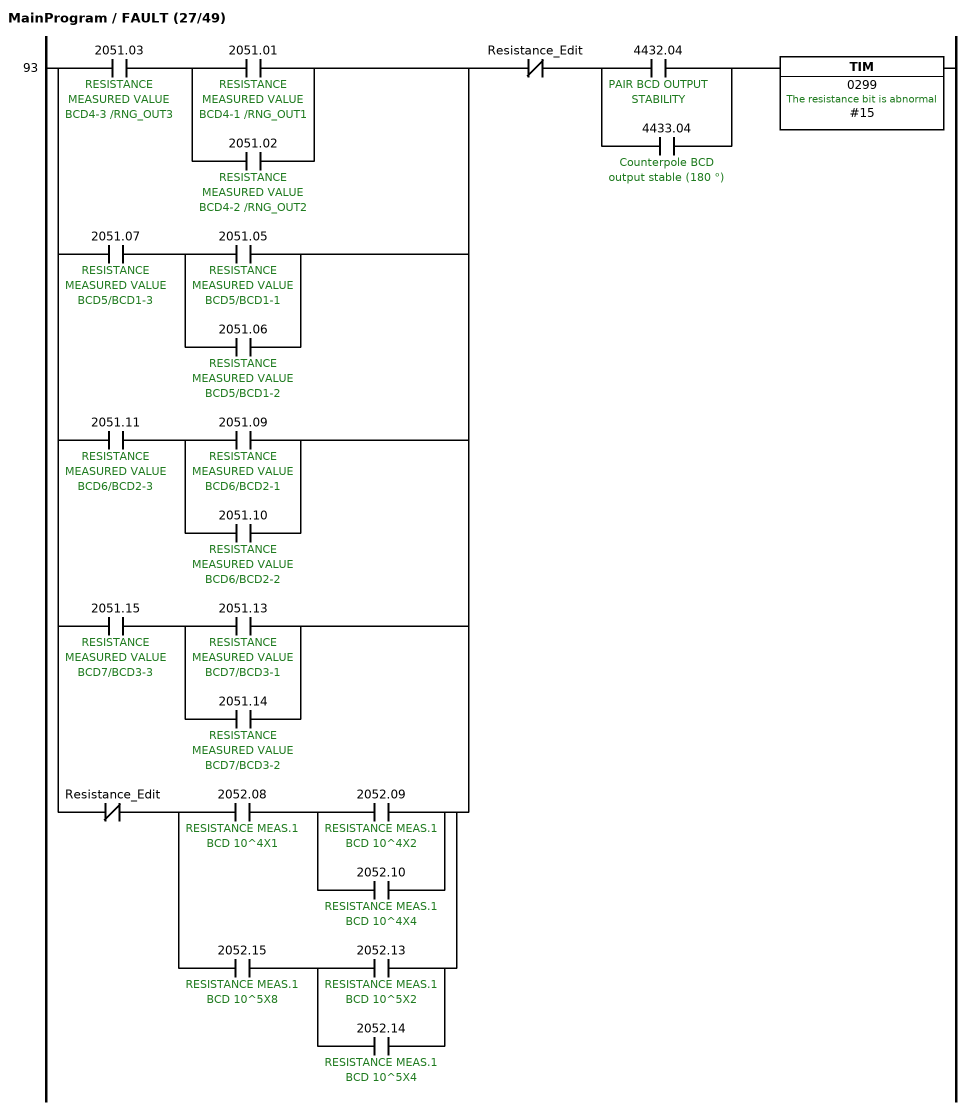
; rung 93
LD 2051.03  ; RESISTANCE MEASURED VALUE BCD4-3 /RNG_OUT3
LD 2051.01  ; RESISTANCE MEASURED VALUE BCD4-1 /RNG_OUT1
OR 2051.02  ; RESISTANCE MEASURED VALUE BCD4-2 /RNG_OUT2
ANDLD
LD 2051.07  ; RESISTANCE MEASURED VALUE BCD5/BCD1-3
LD 2051.05  ; RESISTANCE MEASURED VALUE BCD5/BCD1-1
OR 2051.06  ; RESISTANCE MEASURED VALUE BCD5/BCD1-2
ANDLD
ORLD
LD 2051.11  ; RESISTANCE MEASURED VALUE BCD6/BCD2-3
LD 2051.09  ; RESISTANCE MEASURED VALUE BCD6/BCD2-1
OR 2051.10  ; RESISTANCE MEASURED VALUE BCD6/BCD2-2
ANDLD
ORLD
LD 2051.15  ; RESISTANCE MEASURED VALUE BCD7/BCD3-3
LD 2051.13  ; RESISTANCE MEASURED VALUE BCD7/BCD3-1
OR 2051.14  ; RESISTANCE MEASURED VALUE BCD7/BCD3-2
ANDLD
ORLD
LDNOT Resistance_Edit
LD 2052.08  ; RESISTANCE MEAS.1 BCD 10^4X1
LD 2052.09  ; RESISTANCE MEAS.1 BCD 10^4X2
OR 2052.10  ; RESISTANCE MEAS.1 BCD 10^4X4
ANDLD
LD 2052.15  ; RESISTANCE MEAS.1 BCD 10^5X8
LD 2052.13  ; RESISTANCE MEAS.1 BCD 10^5X2
OR 2052.14  ; RESISTANCE MEAS.1 BCD 10^5X4
ANDLD
ORLD
ANDLD
ORLD
ANDNOT Resistance_Edit
LD 4432.04  ; PAIR BCD OUTPUT STABILITY
OR 4433.04  ; Counterpole BCD output stable (180 °)
ANDLD
TIM 0299 #15  ; The resistance bit is abnormal

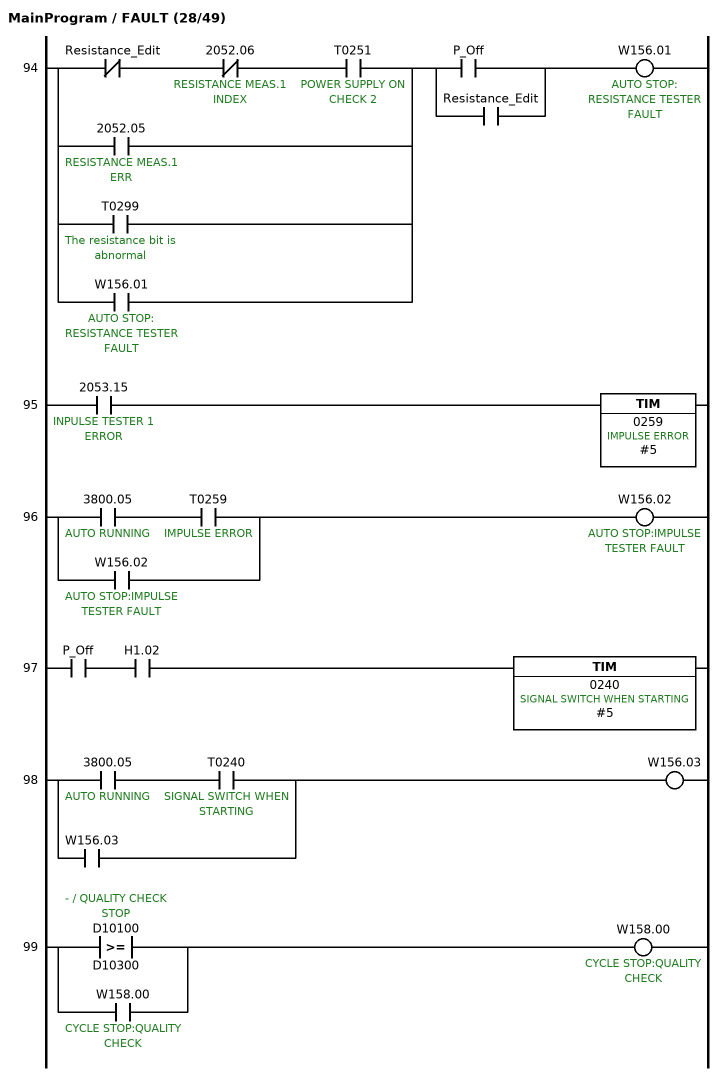
; rung 94
LDNOT Resistance_Edit
ANDNOT 2052.06  ; RESISTANCE MEAS.1 INDEX
AND T0251  ; POWER SUPPLY ON CHECK 2
OR 2052.05  ; RESISTANCE MEAS.1 ERR
OR T0299  ; The resistance bit is abnormal
OR W156.01  ; AUTO STOP:RESISTANCE TESTER FAULT
LD P_Off
OR Resistance_Edit
ANDLD
OUT W156.01  ; AUTO STOP:RESISTANCE TESTER FAULT
; rung 95
LD 2053.15  ; INPULSE TESTER 1 ERROR
TIM 0259 #5  ; IMPULSE ERROR
; rung 96
LD 3800.05  ; AUTO RUNNING
AND T0259  ; IMPULSE ERROR
OR W156.02  ; AUTO STOP:IMPULSE TESTER FAULT
OUT W156.02  ; AUTO STOP:IMPULSE TESTER FAULT
; rung 97
LD P_Off
AND H1.02
TIM 0240 #5  ; SIGNAL SWITCH WHEN STARTING
; rung 98
LD 3800.05  ; AUTO RUNNING
AND T0240  ; SIGNAL SWITCH WHEN STARTING
OR W156.03
OUT W156.03
; rung 99
LD>=L(326) D10100 D10300  ; -, QUALITY CHECK STOP
OR W158.00  ; CYCLE STOP:QUALITY CHECK
OUT W158.00  ; CYCLE STOP:QUALITY CHECK

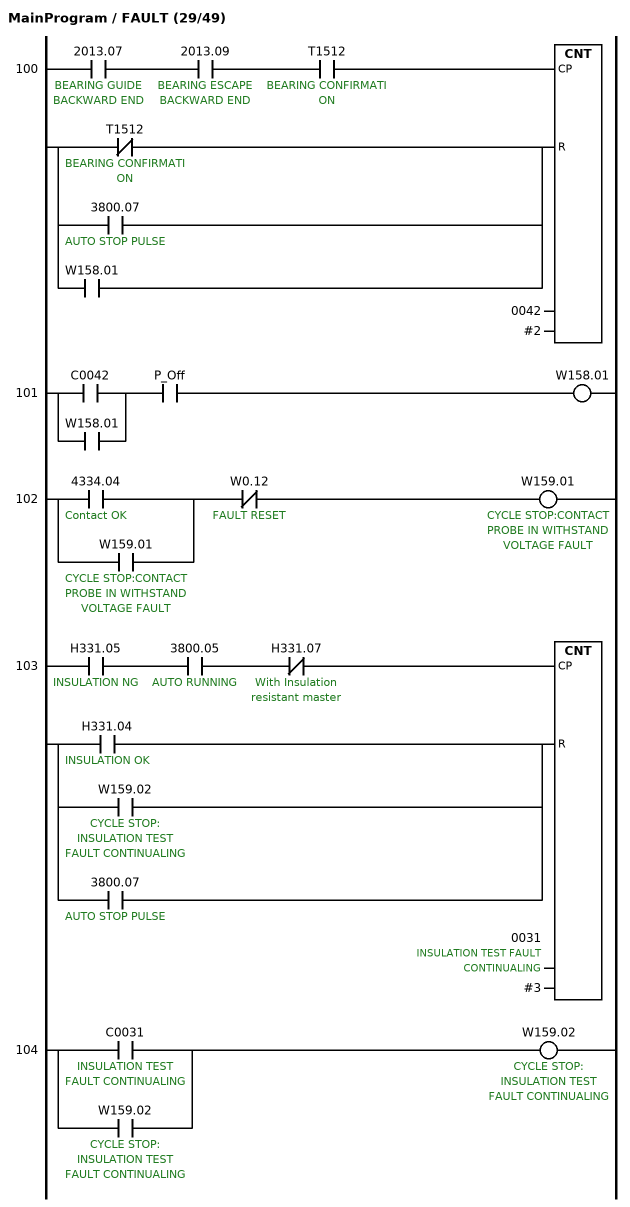
; rung 100
LD 2013.07  ; BEARING GUIDE BACKWARD END
AND 2013.09  ; BEARING ESCAPE BACKWARD END
AND T1512  ; BEARING CONFIRMATION
LDNOT T1512  ; BEARING CONFIRMATION
OR 3800.07  ; AUTO STOP PULSE
OR W158.01
CNT 0042 #2
; rung 101
LD C0042
OR W158.01
AND P_Off
OUT W158.01
; rung 102
LD 4334.04  ; Contact OK
OR W159.01  ; CYCLE STOP:CONTACT PROBE IN WITHSTAND VOLTAGE FAULT
ANDNOT W0.12  ; FAULT RESET
OUT W159.01  ; CYCLE STOP:CONTACT PROBE IN WITHSTAND VOLTAGE FAULT
; rung 103
LD H331.05  ; INSULATION NG
AND 3800.05  ; AUTO RUNNING
ANDNOT H331.07  ; With Insulation resistant master
LD H331.04  ; INSULATION OK
OR W159.02  ; CYCLE STOP:INSULATION TEST FAULT CONTINUALING
OR 3800.07  ; AUTO STOP PULSE
CNT 0031 #3  ; INSULATION TEST FAULT CONTINUALING
; rung 104
LD C0031  ; INSULATION TEST FAULT CONTINUALING
OR W159.02  ; CYCLE STOP:INSULATION TEST FAULT CONTINUALING
OUT W159.02  ; CYCLE STOP:INSULATION TEST FAULT CONTINUALING

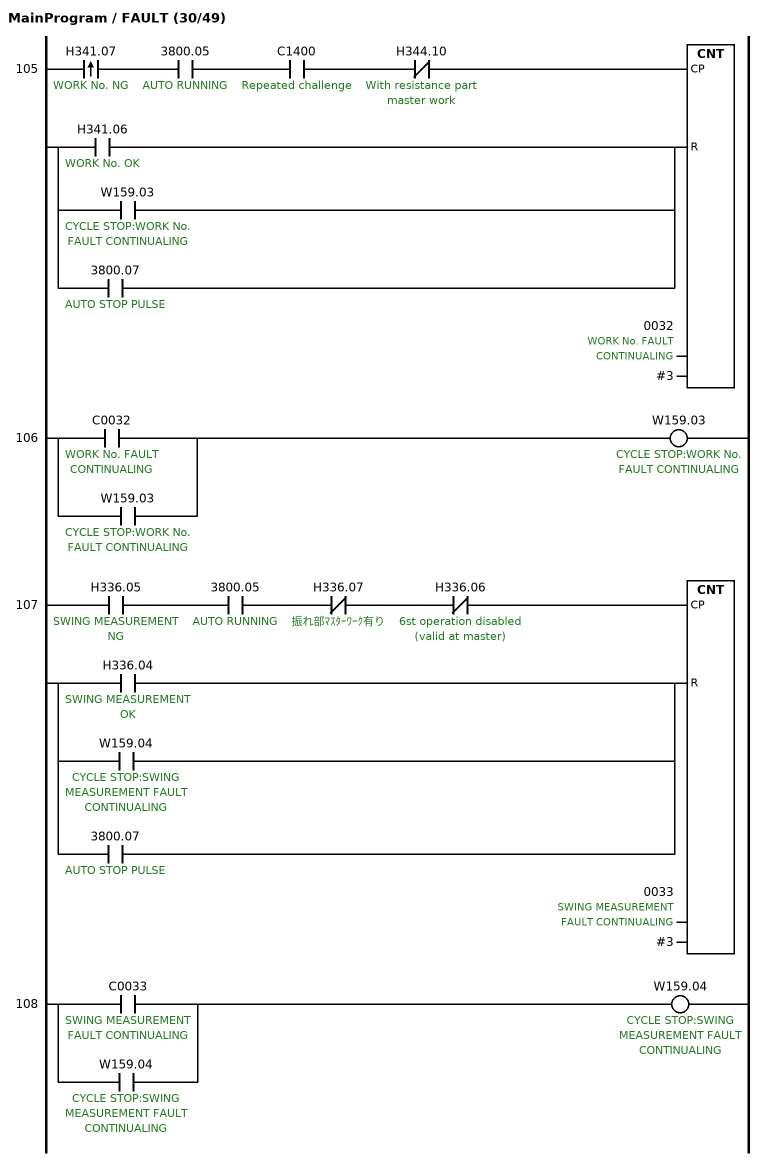
; rung 105
@LD H341.07  ; WORK No. NG
AND 3800.05  ; AUTO RUNNING
AND C1400  ; Repeated challenge
ANDNOT H344.10  ; With resistance part master work
LD H341.06  ; WORK No. OK
OR W159.03  ; CYCLE STOP:WORK No. FAULT CONTINUALING
OR 3800.07  ; AUTO STOP PULSE
CNT 0032 #3  ; WORK No. FAULT CONTINUALING
; rung 106
LD C0032  ; WORK No. FAULT CONTINUALING
OR W159.03  ; CYCLE STOP:WORK No. FAULT CONTINUALING
OUT W159.03  ; CYCLE STOP:WORK No. FAULT CONTINUALING
; rung 107
LD H336.05  ; SWING MEASUREMENT NG
AND 3800.05  ; AUTO RUNNING
ANDNOT H336.07  ; 振れ部ﾏｽﾀｰﾜｰｸ有り
ANDNOT H336.06  ; 6st operation disabled (valid at master)
LD H336.04  ; SWING MEASUREMENT OK
OR W159.04  ; CYCLE STOP:SWING MEASUREMENT FAULT CONTINUALING
OR 3800.07  ; AUTO STOP PULSE
CNT 0033 #3  ; SWING MEASUREMENT FAULT CONTINUALING
; rung 108
LD C0033  ; SWING MEASUREMENT FAULT CONTINUALING
OR W159.04  ; CYCLE STOP:SWING MEASUREMENT FAULT CONTINUALING
OUT W159.04  ; CYCLE STOP:SWING MEASUREMENT FAULT CONTINUALING

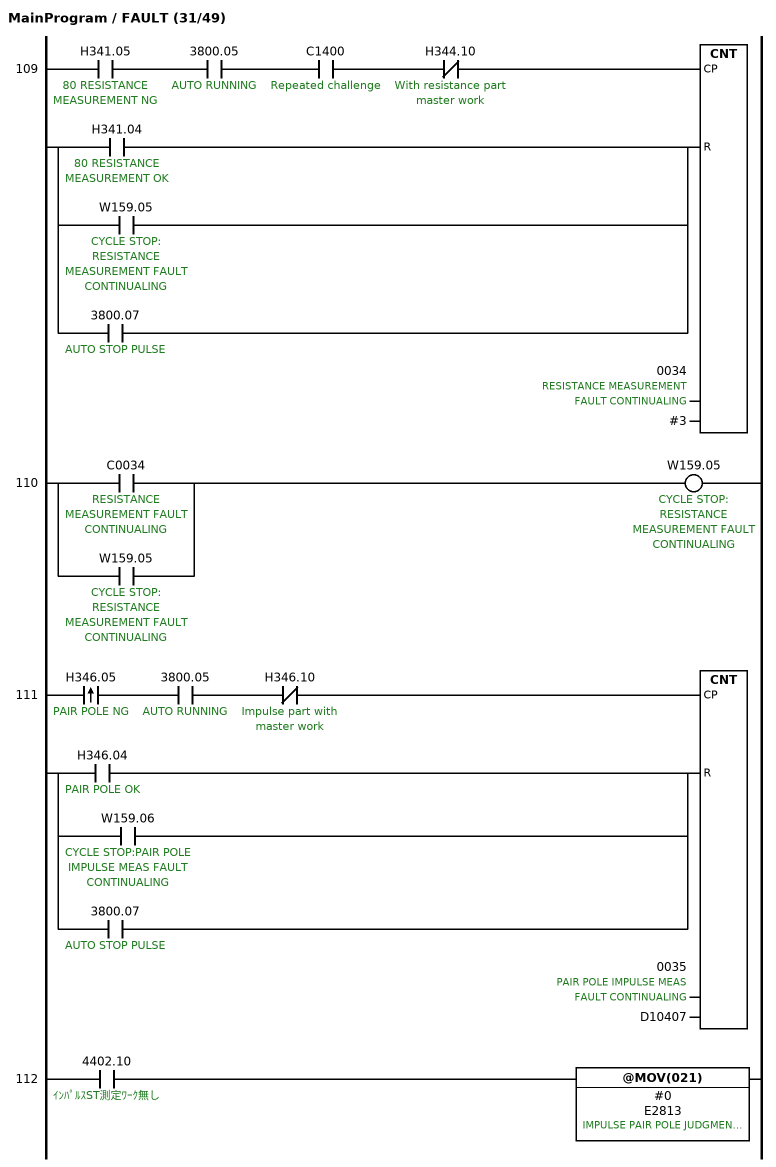
; rung 109
LD H341.05  ; 80 RESISTANCE MEASUREMENT NG
AND 3800.05  ; AUTO RUNNING
AND C1400  ; Repeated challenge
ANDNOT H344.10  ; With resistance part master work
LD H341.04  ; 80 RESISTANCE MEASUREMENT OK
OR W159.05  ; CYCLE STOP:RESISTANCE MEASUREMENT FAULT CONTINUALING
OR 3800.07  ; AUTO STOP PULSE
CNT 0034 #3  ; RESISTANCE MEASUREMENT FAULT CONTINUALING
; rung 110
LD C0034  ; RESISTANCE MEASUREMENT FAULT CONTINUALING
OR W159.05  ; CYCLE STOP:RESISTANCE MEASUREMENT FAULT CONTINUALING
OUT W159.05  ; CYCLE STOP:RESISTANCE MEASUREMENT FAULT CONTINUALING
; rung 111
@LD H346.05  ; PAIR POLE NG
AND 3800.05  ; AUTO RUNNING
ANDNOT H346.10  ; Impulse part with master work
LD H346.04  ; PAIR POLE OK
OR W159.06  ; CYCLE STOP:PAIR POLE IMPULSE MEAS FAULT CONTINUALING
OR 3800.07  ; AUTO STOP PULSE
CNT 0035 D10407  ; PAIR POLE IMPULSE MEAS FAULT CONTINUALING
; rung 112
LD 4402.10  ; ｲﾝﾊﾟﾙｽST測定ﾜｰｸ無し
@MOV(021) #0 E2813  ; IMPULSE PAIR POLE JUDGMENT RESULT (1:OK,2:NG)

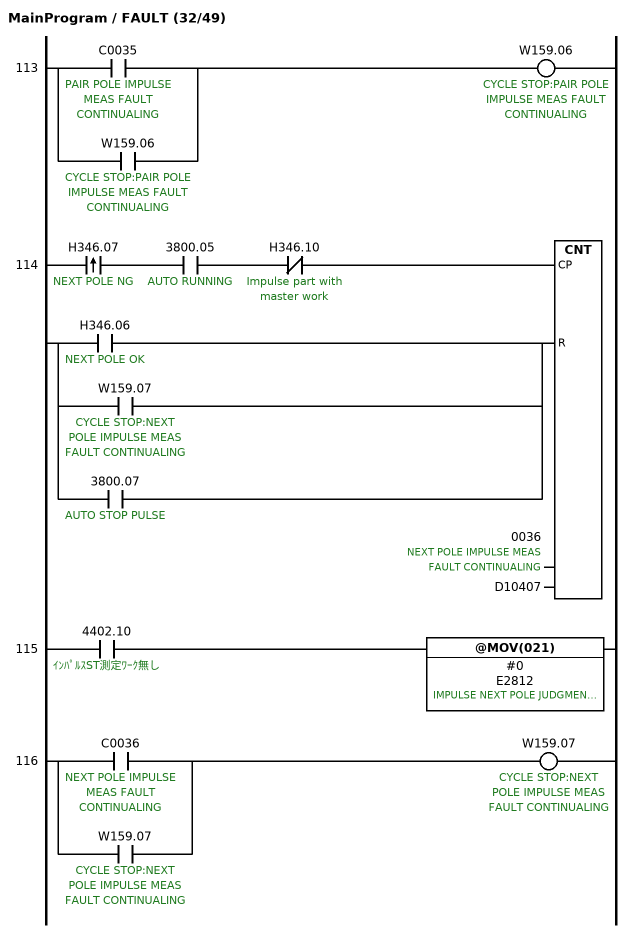
; rung 113
LD C0035  ; PAIR POLE IMPULSE MEAS FAULT CONTINUALING
OR W159.06  ; CYCLE STOP:PAIR POLE IMPULSE MEAS FAULT CONTINUALING
OUT W159.06  ; CYCLE STOP:PAIR POLE IMPULSE MEAS FAULT CONTINUALING
; rung 114
@LD H346.07  ; NEXT POLE NG
AND 3800.05  ; AUTO RUNNING
ANDNOT H346.10  ; Impulse part with master work
LD H346.06  ; NEXT POLE OK
OR W159.07  ; CYCLE STOP:NEXT POLE IMPULSE MEAS FAULT CONTINUALING
OR 3800.07  ; AUTO STOP PULSE
CNT 0036 D10407  ; NEXT POLE IMPULSE MEAS FAULT CONTINUALING
; rung 115
LD 4402.10  ; ｲﾝﾊﾟﾙｽST測定ﾜｰｸ無し
@MOV(021) #0 E2812  ; IMPULSE NEXT POLE JUDGMENT RESULT (1:OK,2:NG)
; rung 116
LD C0036  ; NEXT POLE IMPULSE MEAS FAULT CONTINUALING
OR W159.07  ; CYCLE STOP:NEXT POLE IMPULSE MEAS FAULT CONTINUALING
OUT W159.07  ; CYCLE STOP:NEXT POLE IMPULSE MEAS FAULT CONTINUALING

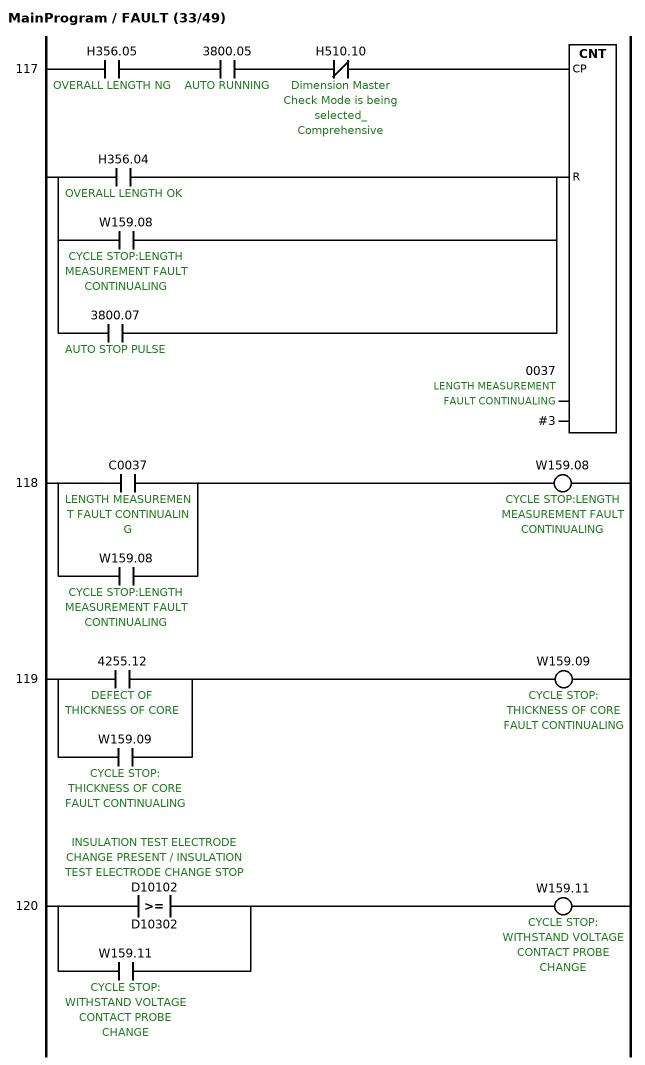
; rung 117
LD H356.05  ; OVERALL LENGTH NG
AND 3800.05  ; AUTO RUNNING
ANDNOT H510.10  ; Dimension Master Check Mode is being selected_Comprehensive
LD H356.04  ; OVERALL LENGTH OK
OR W159.08  ; CYCLE STOP:LENGTH MEASUREMENT FAULT CONTINUALING
OR 3800.07  ; AUTO STOP PULSE
CNT 0037 #3  ; LENGTH MEASUREMENT FAULT CONTINUALING
; rung 118
LD C0037  ; LENGTH MEASUREMENT FAULT CONTINUALING
OR W159.08  ; CYCLE STOP:LENGTH MEASUREMENT FAULT CONTINUALING
OUT W159.08  ; CYCLE STOP:LENGTH MEASUREMENT FAULT CONTINUALING
; rung 119
LD 4255.12  ; DEFECT OF THICKNESS OF CORE
OR W159.09  ; CYCLE STOP:THICKNESS OF CORE FAULT CONTINUALING
OUT W159.09  ; CYCLE STOP:THICKNESS OF CORE FAULT CONTINUALING
; rung 120
LD>=L(326) D10102 D10302  ; INSULATION TEST ELECTRODE CHANGE PRESENT, INSULATION TEST ELECTRODE CHANGE STOP
OR W159.11  ; CYCLE STOP:WITHSTAND VOLTAGE CONTACT PROBE CHANGE
OUT W159.11  ; CYCLE STOP:WITHSTAND VOLTAGE CONTACT PROBE CHANGE

